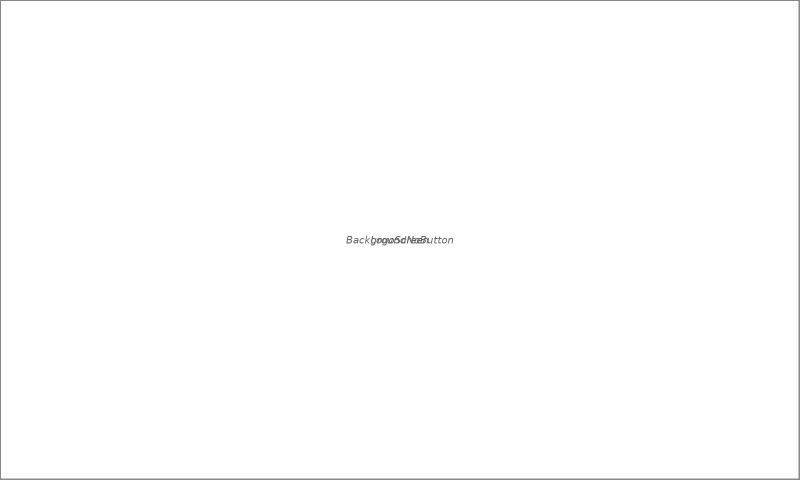
VISUALIZATION StartScreen  // 800x480
    Frame (0,0 800x480)
        shows BackgroundNoButton()
    Frame (0,0 800x480), frame switch variable: GVL_HMI.nStartVisu
        shows LogoScreen()
        shows ParameterScreen()
        shows ManualControl()
END_VISUALIZATION

(* stored: Version 1.1.0.1, ProductVersion 3.1.4024.5
   Visu StartScreen: Id {9c0dfbb2-ead7-41c1-9ffd-e66a861a7940} *)
